# EPICS substitutions: bkhApp/Db/hide/bkhxWRegs.substitutions
file bkhxWReg.template
{
pattern	{                  DESC,       MOD,OFF,  N}
	{       "PLC Interface",BKH$(M)_W1,  0,  1}
	{  "Bus Term Diagnosis",BKH$(M)_W1,  1,  2}
	{ "Watchdog Tmout (ms)",BKH$(M)_W2,  0, 23}
	{      "Watchdog Reset",BKH$(M)_W2,  1, 24}
	{       "Watchdog type",BKH$(M)_W2,  2, 25}
	{     "Modbus TCP mode",BKH$(M)_W2,  3, 26}
}
